PROGRAM MAIN
VAR
END_VAR

POU();

END_PROGRAM

(* stored: Version 1.1.0.1, ProductVersion 3.1.4024.12
   POU MAIN: Id {0df7fef2-dd85-44c0-b78d-5fbef1e7a794}, SpecialFunc None *)
